FUNCTION_BLOCK EK1110

VAR_INPUT
	En				: BOOL;
	iTerminal_ID	: INT;
	ErrorSystem		: POINTER TO ST_ErrorSystem;
END_VAR

VAR_OUTPUT
	EnO		: BOOL;
	bError	: BOOL;
END_VAR

VAR
	InfoData_State	AT %I*	: UINT;
	
	//FB-s
	EK1110_Error	: FB_TerminalError;
END_VAR

(*
* TODO: DONE!
*)
EnO:=En;

//Error FB instance
EK1110_Error(
	En					:= TRUE,
	iTerminal_ID		:= iTerminal_ID,
	bWcState			:= FALSE,
	uiInfoData_State	:= InfoData_State,
	pErrorSystem		:= ErrorSystem,
	bError				=> bError,
);

END_FUNCTION_BLOCK

(* stored: Version 1.1.0.1, ProductVersion 3.1.4024.0
   POU EK1110: Id {b67642f8-ad4b-49aa-ab86-2ce918244b5d}, SpecialFunc None *)
